FUNCTION_BLOCK LrealComparator IMPLEMENTS I_Comparator,I_StepCondition
VAR_INPUT
END_VAR
VAR_OUTPUT
END_VAR
VAR
	uiSelector 		: UINT;
	rInternTarget1 	: REFERENCE TO LREAL;
	rInternTarget2 	: REFERENCE TO LREAL;
	bValue			: BOOL;
END_VAR

IF NOT __ISVALIDREF( rInternTarget1 )
OR NOT __ISVALIDREF( rInternTarget1 )
THEN
	uiSelector := 0;
END_IF 

CASE uiSelector OF

	0:;
		
	10:
		bValue := mEquals(rInternTarget1,rInternTarget2);
		
	20:
		bValue := mGreaterThan(rInternTarget1,rInternTarget2);
	
	30:
		bValue := mLessThan(rInternTarget1,rInternTarget2);
	
	40:
		bValue := mGreaterEquals(rInternTarget1,rInternTarget2);
		
	50:
		bValue := mLessEquals(rInternTarget1,rInternTarget2);
		
END_CASE

{warning 'Eigenschaftenimplementierung hinzufügen'}
PROPERTY getValue : BOOL
GET
getValue := bValue;
END_GET
END_PROPERTY

METHOD mEquals : BOOL;
VAR_INPUT
	rTarget1 : REFERENCE TO LREAL;
	rTarget2 : REFERENCE TO LREAL;
END_VAR
uiSelector := 10;
rInternTarget1 REF= rTarget1;
rInternTarget2 REF= rTarget2;

mEquals := ( rTarget1 = rTarget2 );
END_METHOD

METHOD PUBLIC mGreaterEquals : BOOL
VAR_INPUT
	rTarget1 : REFERENCE TO LREAL;
	rTarget2 : REFERENCE TO LREAL;
END_VAR
uiSelector := 40;
rInternTarget1 REF= rTarget1;
rInternTarget2 REF= rTarget2;

mGreaterEquals := ( rTarget1 >= rTarget2 );
END_METHOD

METHOD mGreaterThan : BOOL;
VAR_INPUT
	rTarget1 : REFERENCE TO LREAL;
	rTarget2 : REFERENCE TO LREAL;
END_VAR
uiSelector := 20;
rInternTarget1 REF= rTarget1;
rInternTarget2 REF= rTarget2;

mGreaterThan := ( rTarget1 >= rTarget2 );
END_METHOD

METHOD mLessEquals : BOOL
VAR_INPUT
	rTarget1 : REFERENCE TO LREAL;
	rTarget2 : REFERENCE TO LREAL;
END_VAR
uiSelector := 50;
rInternTarget1 REF= rTarget1;
rInternTarget2 REF= rTarget2;

mLessEquals := ( rTarget1 <= rTarget2 );
END_METHOD

METHOD mLessThan : BOOL;
VAR_INPUT
	rTarget1 : REFERENCE TO LREAL;
	rTarget2 : REFERENCE TO LREAL;
END_VAR
uiSelector := 30;
rInternTarget1 REF= rTarget1;
rInternTarget2 REF= rTarget2;

mLessThan := ( rTarget1 < rTarget2 );
END_METHOD

{warning 'Eigenschaftenimplementierung hinzufügen'}
PROPERTY setValue : BOOL
SET
bValue := setValue;
END_SET
END_PROPERTY

END_FUNCTION_BLOCK

(* stored: Version 1.1.0.1, ProductVersion 3.1.4024.0
   POU LrealComparator: Id {2e958aad-0ef9-4398-95b3-b78da7119e82}, SpecialFunc None
   Property getValue: Id {d94101d7-2074-4a76-b5aa-3b15557b9eb6}
   Get Get: Id {7ae1ced3-ddda-4bf2-9295-601b95c72942}
   Method mEquals: Id {ffd2e831-e57a-4100-972c-a105e0d81be7}
   Method mGreaterEquals: Id {0d677373-3105-4b7c-824c-f98c1b3af137}
   Method mGreaterThan: Id {53ce0d21-523d-4f73-bd5c-3e6617700c81}
   Method mLessEquals: Id {2f704470-1946-4a75-b673-4eb15855e274}
   Method mLessThan: Id {b968b574-ed4c-467a-a811-6649162c42fc}
   Property setValue: Id {d6bbf76a-b7e8-4f07-a6e2-e0faac8b6802}
   Set Set: Id {2646919f-6395-4d3f-b22b-4bf1ec026f04} *)
